Staubli VAL3: GetProductMess.pgx

program GetProductMess(string x_sMess)
  local num l_nNum
begin
  //生产信息列表
  //专为生产界面


  sMess[0]="---生产日志---"
  sSItem[1]="               "
  if sMess[2]!=x_sMess


    for l_nNum=10 to 3 step -1
      sMess[l_nNum]=sMess[l_nNum-1]
    endFor
    sMess[2]=x_sMess
  endIf
end
